SUBAPPLICATION mapping_Uebung_029 (* LED_DO Blinkende LED *)
  (* Standard: 61499-2 *)
  (* Version 1.0, 2023-10-23, franz *)
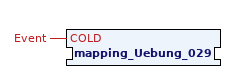
  EVENT_INPUT
    COLD;
  END_EVENT
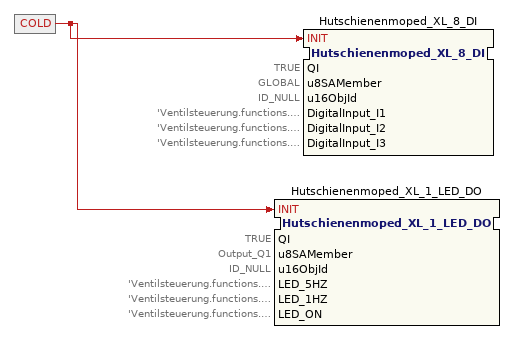
  FBS
    Hutschienenmoped_XL_8_DI : Hutschienenmoped_XL_8_DI(QI := TRUE, u8SAMember := GLOBAL, u16ObjId := ID_NULL, DigitalInput_I1 := 'Ventilsteuerung.functions.DigitalInput_I1', DigitalInput_I2 := 'Ventilsteuerung.functions.DigitalInput_I2', DigitalInput_I3 := 'Ventilsteuerung.functions.DigitalInput_I3');
    Hutschienenmoped_XL_1_LED_DO : Hutschienenmoped_XL_1_LED_DO(QI := TRUE, u8SAMember := Output_Q1, u16ObjId := ID_NULL, LED_5HZ := 'Ventilsteuerung.functions.LED_Q1_5HZ', LED_1HZ := 'Ventilsteuerung.functions.LED_Q1_1HZ', LED_ON := 'Ventilsteuerung.functions.LED_Q1_ON');
  END_FBS
  EVENT_CONNECTIONS
    COLD TO Hutschienenmoped_XL_8_DI.INIT;
    COLD TO Hutschienenmoped_XL_1_LED_DO.INIT;
  END_CONNECTIONS
END_SUBAPPLICATION
